FUNCTION_BLOCK F_TIME_TO_WORD (* convert TIME to WORD *)
  (* Standard: 61131-3; Classification: type conversion function *)
  (* Version 0.0, 2013-08-29, 4DIAC-IDE, 4DIAC-Consortium *)
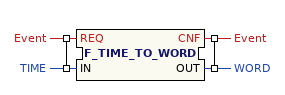
  EVENT_INPUT
    REQ WITH IN; (* Service Request *)
  END_EVENT
  EVENT_OUTPUT
    CNF WITH OUT; (* Confirmation of Requested Service *)
  END_EVENT
  VAR_INPUT
    IN : TIME; (* Event Input Qualifier *)
  END_VAR
  VAR_OUTPUT
    OUT : WORD; (* Event Output Qualifier *)
  END_VAR
END_FUNCTION_BLOCK
